FUNCTION_BLOCK Controller
  (* Standard: 61499-2 *)
  (* Version 0.1, 2017-00-23, hpea485, UOA *)
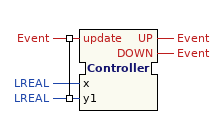
  EVENT_INPUT
    update WITH y1;
  END_EVENT
  EVENT_OUTPUT
    UP;
    DOWN;
  END_EVENT
  VAR_INPUT
    x : LREAL;
    y1 : LREAL;
  END_VAR
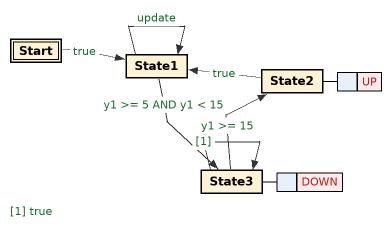
  EC_STATES
    Start;
    State1;
    State2 : -> UP;
    State3 : -> DOWN;
  END_STATES
  EC_TRANSITIONS
    Start TO State1 := true;
    State1 TO State3 := y1 >= 5 AND y1 < 15;
    State1 TO State1 := update;
    State2 TO State1 := true;
    State3 TO State2 := y1 >= 15;
    State3 TO State3 := true;
  END_TRANSITIONS
END_FUNCTION_BLOCK
